(* IEC 61131-3 sources: st-fmt/tests/fixtures/pou, 10 files *)

(* ---- function_block.expected.st ---- *)
FUNCTION_BLOCK FB_Motor
VAR_INPUT
    bStart : BOOL;
END_VAR
VAR
    nState : INT;
END_VAR

IF bStart THEN
    nState := 1;
END_IF

END_FUNCTION_BLOCK

(* ---- function_block.st ---- *)
function_block FB_Motor
var_input
bStart : bool;
end_var
VAR
nState:int;
END_VAR
if bStart then
nState := 1;
end_if;
end_function_block

(* ---- inheritance.expected.st ---- *)
FUNCTION_BLOCK PUBLIC FB_Motor EXTENDS FB_Base IMPLEMENTS I_Motor, I_Resettable
VAR
    n : INT;
END_VAR

n := 1;

END_FUNCTION_BLOCK

INTERFACE I_Motor EXTENDS I_Base
METHOD Run : BOOL
END_METHOD

END_INTERFACE

(* ---- inheritance.st ---- *)
FUNCTION_BLOCK public FB_Motor extends FB_Base implements I_Motor, I_Resettable
VAR
n : INT;
END_VAR
n := 1;
END_FUNCTION_BLOCK
INTERFACE I_Motor extends I_Base
METHOD Run : BOOL
END_METHOD
END_INTERFACE

(* ---- members.expected.st ---- *)
FUNCTION_BLOCK FB_Motor
VAR
    nState : INT;
END_VAR

nState := 0;

METHOD PUBLIC Run : BOOL
VAR_INPUT
    x : INT;
END_VAR

Run := TRUE;
END_METHOD

PROPERTY Speed : REAL
    GET
        Speed := 1.0;
    END_GET
    SET
        ;
    END_SET
END_PROPERTY

ACTION Reset
    nState := 0;
END_ACTION

END_FUNCTION_BLOCK

(* ---- members.st ---- *)
FUNCTION_BLOCK FB_Motor
VAR
nState : INT;
END_VAR
nState := 0;
method public Run : bool
var_input
x : int;
end_var
Run := TRUE;
end_method
property Speed : REAL
get
Speed := 1.0;
end_get
set
;
end_set
end_property
action Reset
nState := 0;
end_action
END_FUNCTION_BLOCK

(* ---- separation.expected.st ---- *)
{attribute 'pack_mode':='1'}
FUNCTION_BLOCK FB_First
n := 1;

END_FUNCTION_BLOCK

// documents the second block
FUNCTION_BLOCK FB_Second
n := 2;

END_FUNCTION_BLOCK

INTERFACE I_Empty
END_INTERFACE

(* ---- separation.st ---- *)
{attribute 'pack_mode':='1'}
FUNCTION_BLOCK FB_First
n := 1;
END_FUNCTION_BLOCK
// documents the second block
FUNCTION_BLOCK FB_Second

n := 2;

END_FUNCTION_BLOCK
INTERFACE I_Empty
END_INTERFACE

(* ---- function_and_program.expected.st ---- *)
FUNCTION Add : INT
VAR_INPUT
    a : INT;
    b : INT;
END_VAR

Add := a + b;

END_FUNCTION

PROGRAM Main
VAR
    x : INT;
END_VAR

x := Add(1, 2);

END_PROGRAM

(* ---- function_and_program.st ---- *)
function Add : int
var_input
a : int;
b : int;
end_var
Add := a + b;
end_function
PROGRAM Main
VAR
x : INT;
END_VAR
x := Add(1, 2);
END_PROGRAM
